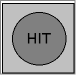
VISUALIZATION FloorPanel  // 76x75
    Rectangle (2,3 72x70)
    Ellipse (12,12 54x53), "HIT", colour toggle: (m_Input_LAMP) <> 0
        tap m_Input_BUTTON
END_VISUALIZATION

(* stored: Version 1.1.0.1, ProductVersion 3.1.4022.12
   Visu FloorPanel: Id {73340785-3dcb-4275-b909-40d06e6623b5} *)
